(* Logix 5000 project; controller R1USB70001_CWRU_GRID_20120217 vendor 1 type 14 code 54 rev 19.11; software revision 19.01; part 2 of 3 *)
(* tags used below, declared in another part *)
   COM_TO_GRID_CLOSE_FAIL : BOOL;
   COM_TO_GRID_CLOSE_FAIL_THRESH : REAL;
   COM_TO_GRID_CLOSE_PROXY : BOOL;
   COM_TO_GRID_CLOSED : BOOL;
   COM_TO_GRID_COMMAND_CHANGED : BOOL;
   COM_TO_GRID_COMMAND_CHANGED_TIMER : TIMER;
   COM_TO_GRID_CURRENT : REAL;
   COM_TO_GRID_INT_REQ_CLOSE : BOOL;
   COM_TO_GRID_INT_REQ_CONNECT : BOOL;
   COM_TO_GRID_OPEN_FAIL : BOOL;
   COM_TO_GRID_OPEN_FAIL_THRESH : REAL;
   COM_TO_GRID_REQ_CLOSE : BOOL;
   COM_TO_GRID_REQ_CONNECT : BOOL;
   COM_TO_GRID_REQ_DISCONNECT : BOOL;
   COM_TO_GRID_REQ_OPEN : BOOL;
   COM_TO_SC_CLOSE_FAIL : BOOL;
   COM_TO_SC_CLOSE_FAIL_THRESH : REAL;
   COM_TO_SC_CLOSE_PROXY : BOOL;
   COM_TO_SC_CLOSED : BOOL;
   COM_TO_SC_COMMAND_CHANGED : BOOL;
   COM_TO_SC_COMMAND_CHANGED_TIMER : TIMER;
   COM_TO_SC_INT_REQ_CLOSE : BOOL;
   COM_TO_SC_INT_REQ_CONNECT : BOOL;
   COM_TO_SC_OPEN_FAIL : BOOL;
   COM_TO_SC_OPEN_FAIL_THRESH : REAL;
   COM_TO_SC_REQ_CLOSE : BOOL;
   COM_TO_SC_REQ_CONNECT : BOOL;
   COM_TO_SC_REQ_DISCONNECT : BOOL;
   COM_TO_SC_REQ_OPEN : BOOL;
   COM_TO_SF_CLOSE_FAIL : BOOL;
   COM_TO_SF_CLOSE_FAIL_THRESH : REAL;
   COM_TO_SF_CLOSE_PROXY : BOOL;
   COM_TO_SF_CLOSED : BOOL;
   COM_TO_SF_COMMAND_CHANGED : BOOL;
   COM_TO_SF_COMMAND_CHANGED_TIMER : TIMER;
   COM_TO_SF_INT_REQ_CLOSE : BOOL;
   COM_TO_SF_INT_REQ_CONNECT : BOOL;
   COM_TO_SF_OPEN_FAIL : BOOL;
   COM_TO_SF_OPEN_FAIL_THRESH : REAL;
   COM_TO_SF_REQ_CLOSE : BOOL;
   COM_TO_SF_REQ_CONNECT : BOOL;
   COM_TO_SF_REQ_DISCONNECT : BOOL;
   COM_TO_SF_REQ_OPEN : BOOL;
   COM_TO_WF_CLOSE_FAIL : BOOL;
   COM_TO_WF_CLOSE_FAIL_THRESH : REAL;
   COM_TO_WF_CLOSE_PROXY : BOOL;
   COM_TO_WF_CLOSED : BOOL;
   COM_TO_WF_COMMAND_CHANGED : BOOL;
   COM_TO_WF_COMMAND_CHANGED_TIMER : TIMER;
   COM_TO_WF_INT_REQ_CLOSE : BOOL;
   COM_TO_WF_INT_REQ_CONNECT : BOOL;
   COM_TO_WF_OPEN_FAIL : BOOL;
   COM_TO_WF_OPEN_FAIL_THRESH : REAL;
   COM_TO_WF_REQ_CLOSE : BOOL;
   COM_TO_WF_REQ_CONNECT : BOOL;
   COM_TO_WF_REQ_DISCONNECT : BOOL;
   COM_TO_WF_REQ_OPEN : BOOL;
   COM_TO_WT_CLOSE_FAIL : BOOL;
   COM_TO_WT_CLOSE_FAIL_THRESH : REAL;
   COM_TO_WT_CLOSE_PROXY : BOOL;
   COM_TO_WT_CLOSED : BOOL;
   COM_TO_WT_COMMAND_CHANGED : BOOL;
   COM_TO_WT_COMMAND_CHANGED_TIMER : TIMER;
   COM_TO_WT_INT_REQ_CLOSE : BOOL;
   COM_TO_WT_INT_REQ_CONNECT : BOOL;
   COM_TO_WT_OPEN_FAIL : BOOL;
   COM_TO_WT_OPEN_FAIL_THRESH : REAL;
   COM_TO_WT_REQ_CLOSE : BOOL;
   COM_TO_WT_REQ_CONNECT : BOOL;
   COM_TO_WT_REQ_DISCONNECT : BOOL;
   COM_TO_WT_REQ_OPEN : BOOL;
   IND_TO_SC_CLOSE_FAIL : BOOL;
   IND_TO_SC_CLOSE_PROXY : BOOL;
   IND_TO_SC_CLOSED : BOOL;
   IND_TO_SC_COMMAND_CHANGED : BOOL;
   IND_TO_SC_COMMAND_CHANGED_TIMER : TIMER;
   IND_TO_SC_INT_REQ_CLOSE : BOOL;
   IND_TO_SC_INT_REQ_CONNECT : BOOL;
   IND_TO_SC_OPEN_FAIL : BOOL;
   IND_TO_SC_REQ_CLOSE : BOOL;
   IND_TO_SC_REQ_CONNECT : BOOL;
   IND_TO_SC_REQ_DISCONNECT : BOOL;
   IND_TO_SC_REQ_OPEN : BOOL;
   IND_TO_SF_CLOSE_FAIL : BOOL;
   IND_TO_SF_CLOSE_FAIL_THRESH : REAL;
   IND_TO_SF_CLOSE_PROXY : BOOL;
   IND_TO_SF_CLOSED : BOOL;
   IND_TO_SF_COMMAND_CHANGED : BOOL;
   IND_TO_SF_COMMAND_CHANGED_TIMER : TIMER;
   IND_TO_SF_INT_REQ_CLOSE : BOOL;
   IND_TO_SF_INT_REQ_CONNECT : BOOL;
   IND_TO_SF_OPEN_FAIL : BOOL;
   IND_TO_SF_OPEN_FAIL_THRESH : REAL;
   IND_TO_SF_REQ_CLOSE : BOOL;
   IND_TO_SF_REQ_CONNECT : BOOL;
   IND_TO_SF_REQ_DISCONNECT : BOOL;
   IND_TO_SF_REQ_OPEN : BOOL;
   IND_TO_WT_CLOSE_FAIL : BOOL;
   IND_TO_WT_CLOSE_FAIL_THRESH : REAL;
   IND_TO_WT_CLOSED : BOOL;
   IND_TO_WT_COMMAND_CHANGED : BOOL;
   IND_TO_WT_COMMAND_CHANGED_TIMER : TIMER;
   IND_TO_WT_INT_REQ_CONNECT : BOOL;
   IND_TO_WT_OPEN_FAIL : BOOL;
   IND_TO_WT_OPEN_FAIL_THRESH : REAL;
   IND_TO_WT_REQ_CLOSE : BOOL;
   IND_TO_WT_REQ_CONNECT : BOOL;
   IND_TO_WT_REQ_OPEN : BOOL;
   SC_TO_COM_CURRENT : REAL;
   SC_TO_GRID_CLOSE_FAIL : BOOL;
   SC_TO_GRID_CLOSE_FAIL_THRESH : REAL;
   SC_TO_GRID_CLOSE_PROXY : BOOL;
   SC_TO_GRID_CLOSED : BOOL;
   SC_TO_GRID_COMMAND_CHANGED : BOOL;
   SC_TO_GRID_COMMAND_CHANGED_TIMER : TIMER;
   SC_TO_GRID_CURRENT : REAL;
   SC_TO_GRID_INT_REQ_CLOSE : BOOL;
   SC_TO_GRID_INT_REQ_CONNECT : BOOL;
   SC_TO_GRID_OPEN_FAIL : BOOL;
   SC_TO_GRID_OPEN_FAIL_THRESH : REAL;
   SC_TO_GRID_REQ_CLOSE : BOOL;
   SC_TO_GRID_REQ_CONNECT : BOOL;
   SC_TO_GRID_REQ_DISCONNECT : BOOL;
   SC_TO_GRID_REQ_OPEN : BOOL;
   SC_TO_IND_CLOSE_FAIL_THRESH : REAL;
   SC_TO_IND_CURRENT : REAL;
   SC_TO_IND_OPEN_FAIL_THRESH : REAL;
   SF_TO_COM_CURRENT : REAL;
   SF_TO_GRID_CLOSE_FAIL : BOOL;
   SF_TO_GRID_CLOSE_FAIL_THRESH : REAL;
   SF_TO_GRID_CLOSE_PROXY : BOOL;
   SF_TO_GRID_CLOSED : BOOL;
   SF_TO_GRID_COMMAND_CHANGED : BOOL;
   SF_TO_GRID_COMMAND_CHANGED_TIMER : TIMER;
   SF_TO_GRID_CURRENT : REAL;
   SF_TO_GRID_INT_REQ_CLOSE : BOOL;
   SF_TO_GRID_INT_REQ_CONNECT : BOOL;
   SF_TO_GRID_OPEN_FAIL : BOOL;
   SF_TO_GRID_OPEN_FAIL_THRESH : REAL;
   SF_TO_GRID_REQ_CLOSE : BOOL;
   SF_TO_GRID_REQ_CONNECT : BOOL;
   SF_TO_GRID_REQ_DISCONNECT : BOOL;
   SF_TO_GRID_REQ_OPEN : BOOL;
   SF_TO_IND_CURRENT : REAL;
   WF_TO_COM_CURRENT : REAL;
   WF_TO_GRID_CLOSE_FAIL : BOOL;
   WF_TO_GRID_CLOSE_FAIL_THRESH : REAL;
   WF_TO_GRID_CLOSE_PROXY : BOOL;
   WF_TO_GRID_CLOSED : BOOL;
   WF_TO_GRID_COMMAND_CHANGED : BOOL;
   WF_TO_GRID_COMMAND_CHANGED_TIMER : TIMER;
   WF_TO_GRID_CURRENT : REAL;
   WF_TO_GRID_INT_REQ_CLOSE : BOOL;
   WF_TO_GRID_INT_REQ_CONNECT : BOOL;
   WF_TO_GRID_OPEN_FAIL : BOOL;
   WF_TO_GRID_OPEN_FAIL_THRESH : REAL;
   WF_TO_GRID_REQ_CLOSE : BOOL;
   WF_TO_GRID_REQ_CONNECT : BOOL;
   WF_TO_GRID_REQ_DISCONNECT : BOOL;
   WF_TO_GRID_REQ_OPEN : BOOL;
   WT_TO_COM_CURRENT : REAL;
   WT_TO_GRID_CLOSE_FAIL : BOOL;
   WT_TO_GRID_CLOSE_FAIL_THRESH : REAL;
   WT_TO_GRID_CLOSE_PROXY : BOOL;
   WT_TO_GRID_CLOSED : BOOL;
   WT_TO_GRID_COMMAND_CHANGED : BOOL;
   WT_TO_GRID_COMMAND_CHANGED_TIMER : TIMER;
   WT_TO_GRID_CURRENT : REAL;
   WT_TO_GRID_INT_REQ_CLOSE : BOOL;
   WT_TO_GRID_INT_REQ_CONNECT : BOOL;
   WT_TO_GRID_OPEN_FAIL : BOOL;
   WT_TO_GRID_OPEN_FAIL_THRESH : REAL;
   WT_TO_GRID_REQ_CLOSE : BOOL;
   WT_TO_GRID_REQ_CONNECT : BOOL;
   WT_TO_GRID_REQ_DISCONNECT : BOOL;
   WT_TO_GRID_REQ_OPEN : BOOL;
   WT_TO_IND_CURRENT : REAL;
   CL_GP_GD_CS : ALIAS FOR ACNR_GP_SC_N2:15:O.1;
   CL_GP_SC_CS : ALIAS FOR ACNR_GP_SC_N2:15:O.5;
   CL_GP_SF_CS : ALIAS FOR ACNR_GP_SC_N2:15:O.4;
   CL_GP_WF_CS : ALIAS FOR ACNR_GP_SC_N2:15:O.2;
   CL_GP_WT_CS : ALIAS FOR ACNR_GP_SC_N2:15:O.3;
   IL_GP_SC_CS : ALIAS FOR ACNR_GP_SC_N2:16:O.2;
   IL_GP_SF_CS : ALIAS FOR ACNR_GP_SC_N2:16:O.1;
   SC_GP_GD_CS : ALIAS FOR ACNR_GP_SC_N2:14:O.2;
   SF_GP_GD_CS : ALIAS FOR ACNR_GP_SC_N2:14:O.0;
   WF_GP_GD_CS : ALIAS FOR ACNR_GP_SC_N2:13:O.3;
   WT_GP_GD_CS : ALIAS FOR ACNR_GP_SC_N2:13:O.5;
(* MainProgram, continued *)

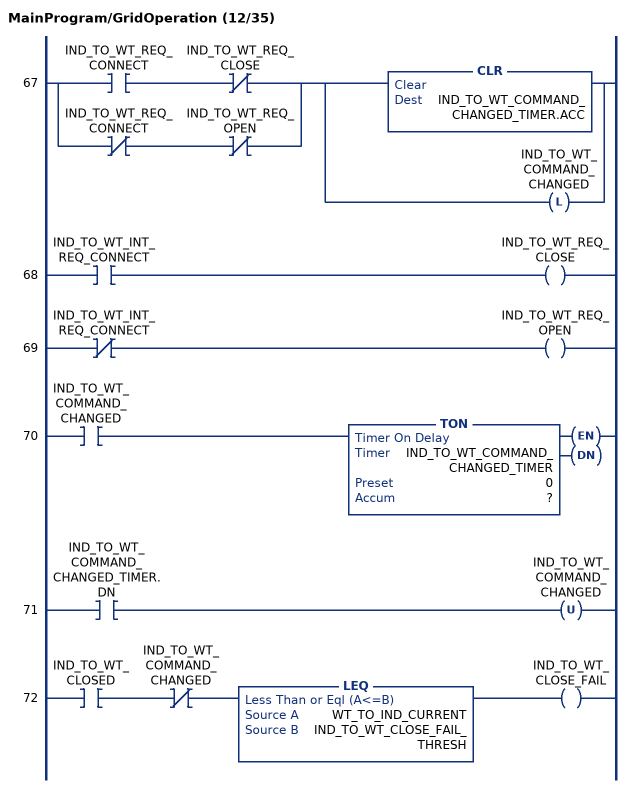
   [picture p24: MainProgram/GridOperation rungs 67-72]
   67: [XIC(IND_TO_WT_REQ_CONNECT) XIO(IND_TO_WT_REQ_CLOSE) ,XIO(IND_TO_WT_REQ_CONNECT) XIO(IND_TO_WT_REQ_OPEN) ][CLR(IND_TO_WT_COMMAND_CHANGED_TIMER.ACC) ,OTL(IND_TO_WT_COMMAND_CHANGED) ];
   68: XIC(IND_TO_WT_INT_REQ_CONNECT)OTE(IND_TO_WT_REQ_CLOSE);
   69: XIO(IND_TO_WT_INT_REQ_CONNECT)OTE(IND_TO_WT_REQ_OPEN);
   70: XIC(IND_TO_WT_COMMAND_CHANGED)TON(IND_TO_WT_COMMAND_CHANGED_TIMER,?,?);
   71: XIC(IND_TO_WT_COMMAND_CHANGED_TIMER.DN)OTU(IND_TO_WT_COMMAND_CHANGED);
   72: XIC(IND_TO_WT_CLOSED)XIO(IND_TO_WT_COMMAND_CHANGED)LEQ(WT_TO_IND_CURRENT,IND_TO_WT_CLOSE_FAIL_THRESH)OTE(IND_TO_WT_CLOSE_FAIL);
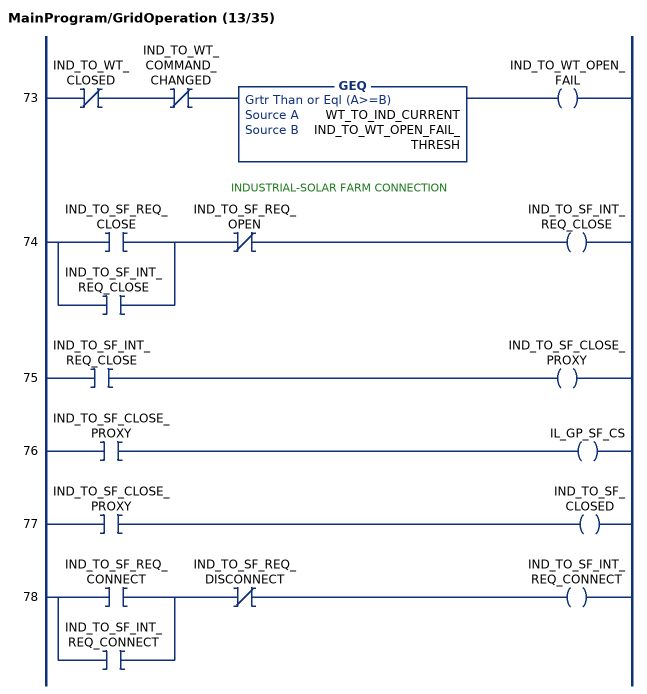
   73: XIO(IND_TO_WT_CLOSED)XIO(IND_TO_WT_COMMAND_CHANGED)GEQ(WT_TO_IND_CURRENT,IND_TO_WT_OPEN_FAIL_THRESH)OTE(IND_TO_WT_OPEN_FAIL);
   // INDUSTRIAL-SOLAR FARM CONNECTION
   74: [XIC(IND_TO_SF_REQ_CLOSE) ,XIC(IND_TO_SF_INT_REQ_CLOSE) ]XIO(IND_TO_SF_REQ_OPEN)OTE(IND_TO_SF_INT_REQ_CLOSE);
   75: XIC(IND_TO_SF_INT_REQ_CLOSE)OTE(IND_TO_SF_CLOSE_PROXY);
   76: XIC(IND_TO_SF_CLOSE_PROXY)OTE(IL_GP_SF_CS);
   77: XIC(IND_TO_SF_CLOSE_PROXY)OTE(IND_TO_SF_CLOSED);
   78: [XIC(IND_TO_SF_REQ_CONNECT) ,XIC(IND_TO_SF_INT_REQ_CONNECT) ]XIO(IND_TO_SF_REQ_DISCONNECT)OTE(IND_TO_SF_INT_REQ_CONNECT);
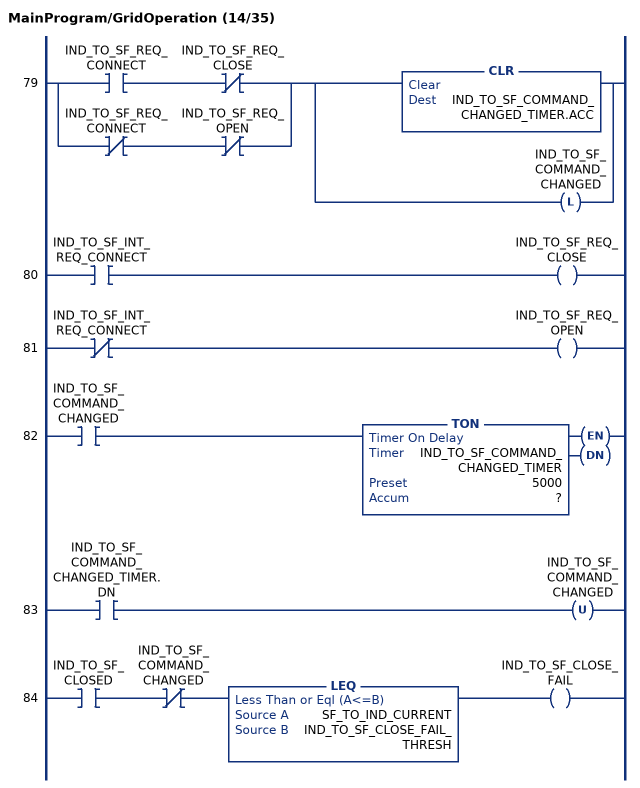
   79: [XIC(IND_TO_SF_REQ_CONNECT) XIO(IND_TO_SF_REQ_CLOSE) ,XIO(IND_TO_SF_REQ_CONNECT) XIO(IND_TO_SF_REQ_OPEN) ][CLR(IND_TO_SF_COMMAND_CHANGED_TIMER.ACC) ,OTL(IND_TO_SF_COMMAND_CHANGED) ];
   80: XIC(IND_TO_SF_INT_REQ_CONNECT)OTE(IND_TO_SF_REQ_CLOSE);
   81: XIO(IND_TO_SF_INT_REQ_CONNECT)OTE(IND_TO_SF_REQ_OPEN);
   82: XIC(IND_TO_SF_COMMAND_CHANGED)TON(IND_TO_SF_COMMAND_CHANGED_TIMER,?,?);
   83: XIC(IND_TO_SF_COMMAND_CHANGED_TIMER.DN)OTU(IND_TO_SF_COMMAND_CHANGED);
   84: XIC(IND_TO_SF_CLOSED)XIO(IND_TO_SF_COMMAND_CHANGED)LEQ(SF_TO_IND_CURRENT,IND_TO_SF_CLOSE_FAIL_THRESH)OTE(IND_TO_SF_CLOSE_FAIL);
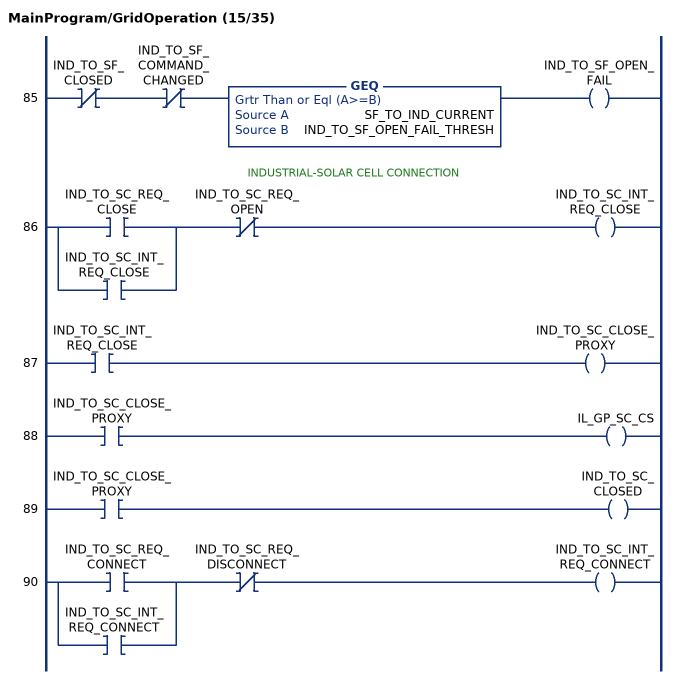
   85: XIO(IND_TO_SF_CLOSED)XIO(IND_TO_SF_COMMAND_CHANGED)GEQ(SF_TO_IND_CURRENT,IND_TO_SF_OPEN_FAIL_THRESH)OTE(IND_TO_SF_OPEN_FAIL);
   // INDUSTRIAL-SOLAR CELL CONNECTION
   86: [XIC(IND_TO_SC_REQ_CLOSE) ,XIC(IND_TO_SC_INT_REQ_CLOSE) ]XIO(IND_TO_SC_REQ_OPEN)OTE(IND_TO_SC_INT_REQ_CLOSE);
   87: XIC(IND_TO_SC_INT_REQ_CLOSE)OTE(IND_TO_SC_CLOSE_PROXY);
   88: XIC(IND_TO_SC_CLOSE_PROXY)OTE(IL_GP_SC_CS);
   89: XIC(IND_TO_SC_CLOSE_PROXY)OTE(IND_TO_SC_CLOSED);
   90: [XIC(IND_TO_SC_REQ_CONNECT) ,XIC(IND_TO_SC_INT_REQ_CONNECT) ]XIO(IND_TO_SC_REQ_DISCONNECT)OTE(IND_TO_SC_INT_REQ_CONNECT);
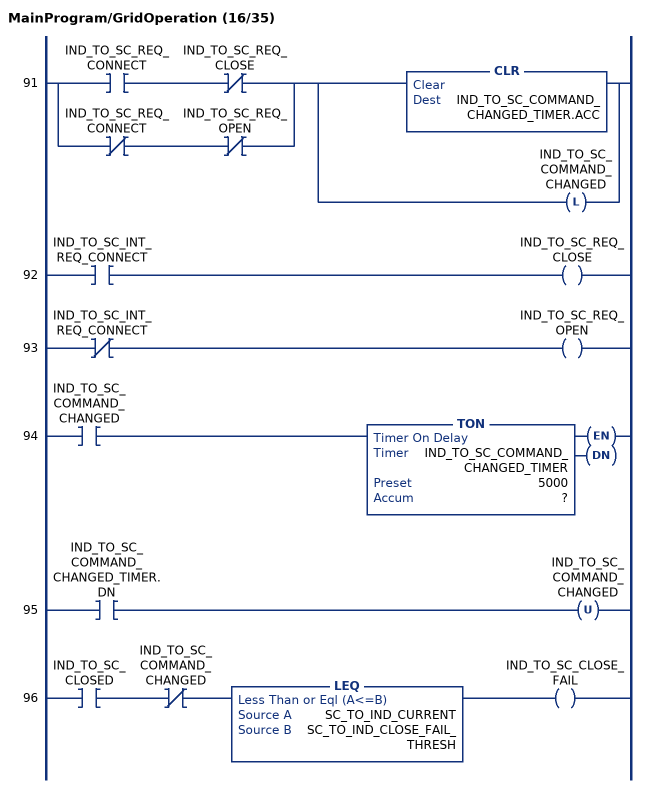
   91: [XIC(IND_TO_SC_REQ_CONNECT) XIO(IND_TO_SC_REQ_CLOSE) ,XIO(IND_TO_SC_REQ_CONNECT) XIO(IND_TO_SC_REQ_OPEN) ][CLR(IND_TO_SC_COMMAND_CHANGED_TIMER.ACC) ,OTL(IND_TO_SC_COMMAND_CHANGED) ];
   92: XIC(IND_TO_SC_INT_REQ_CONNECT)OTE(IND_TO_SC_REQ_CLOSE);
   93: XIO(IND_TO_SC_INT_REQ_CONNECT)OTE(IND_TO_SC_REQ_OPEN);
   94: XIC(IND_TO_SC_COMMAND_CHANGED)TON(IND_TO_SC_COMMAND_CHANGED_TIMER,?,?);
   95: XIC(IND_TO_SC_COMMAND_CHANGED_TIMER.DN)OTU(IND_TO_SC_COMMAND_CHANGED);
   96: XIC(IND_TO_SC_CLOSED)XIO(IND_TO_SC_COMMAND_CHANGED)LEQ(SC_TO_IND_CURRENT,SC_TO_IND_CLOSE_FAIL_THRESH)OTE(IND_TO_SC_CLOSE_FAIL);
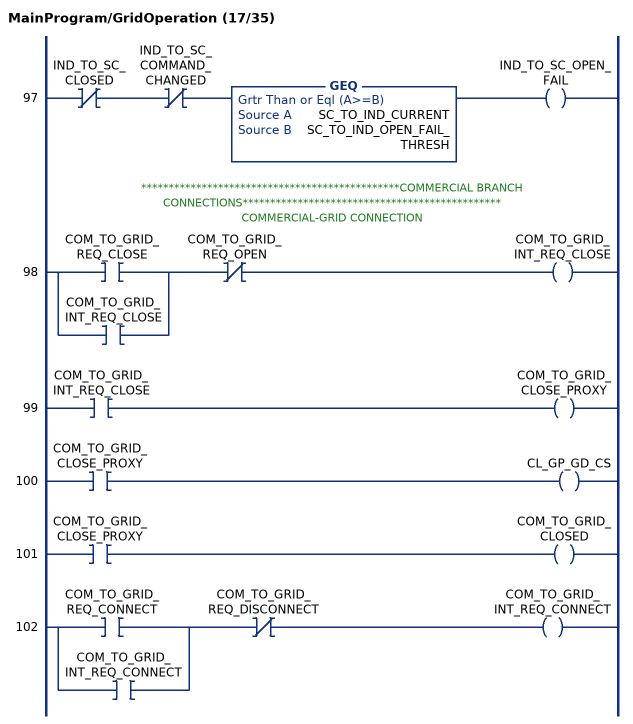
   97: XIO(IND_TO_SC_CLOSED)XIO(IND_TO_SC_COMMAND_CHANGED)GEQ(SC_TO_IND_CURRENT,SC_TO_IND_OPEN_FAIL_THRESH)OTE(IND_TO_SC_OPEN_FAIL);
   // ***********************************************COMMERCIAL BRANCH CONNECTIONS***********************************************
   // COMMERCIAL-GRID CONNECTION
   98: [XIC(COM_TO_GRID_REQ_CLOSE) ,XIC(COM_TO_GRID_INT_REQ_CLOSE) ]XIO(COM_TO_GRID_REQ_OPEN)OTE(COM_TO_GRID_INT_REQ_CLOSE);
   99: XIC(COM_TO_GRID_INT_REQ_CLOSE)OTE(COM_TO_GRID_CLOSE_PROXY);
   100: XIC(COM_TO_GRID_CLOSE_PROXY)OTE(CL_GP_GD_CS);
   101: XIC(COM_TO_GRID_CLOSE_PROXY)OTE(COM_TO_GRID_CLOSED);
   102: [XIC(COM_TO_GRID_REQ_CONNECT) ,XIC(COM_TO_GRID_INT_REQ_CONNECT) ]XIO(COM_TO_GRID_REQ_DISCONNECT)OTE(COM_TO_GRID_INT_REQ_CONNECT);
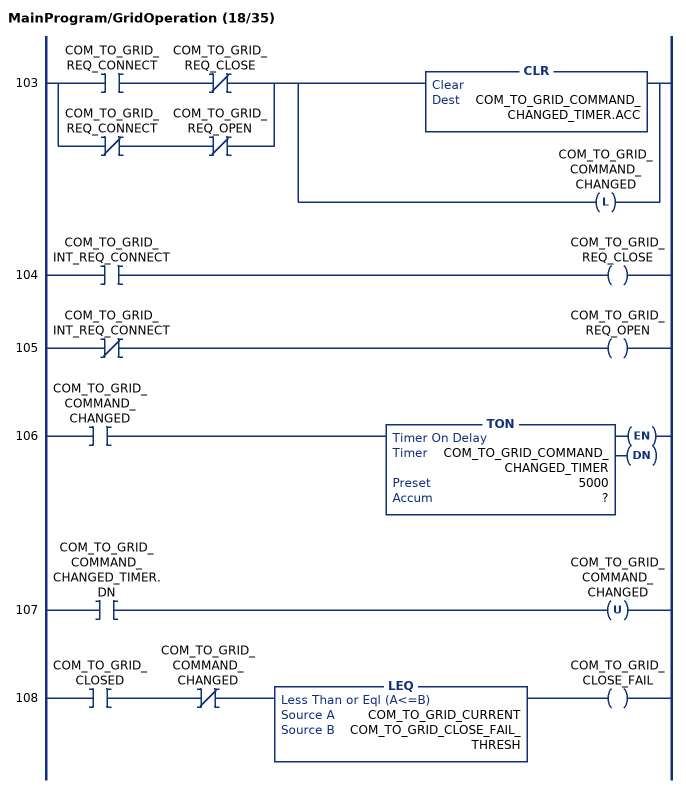
   103: [XIC(COM_TO_GRID_REQ_CONNECT) XIO(COM_TO_GRID_REQ_CLOSE) ,XIO(COM_TO_GRID_REQ_CONNECT) XIO(COM_TO_GRID_REQ_OPEN) ][CLR(COM_TO_GRID_COMMAND_CHANGED_TIMER.ACC) ,OTL(COM_TO_GRID_COMMAND_CHANGED) ];
   104: XIC(COM_TO_GRID_INT_REQ_CONNECT)OTE(COM_TO_GRID_REQ_CLOSE);
   105: XIO(COM_TO_GRID_INT_REQ_CONNECT)OTE(COM_TO_GRID_REQ_OPEN);
   106: XIC(COM_TO_GRID_COMMAND_CHANGED)TON(COM_TO_GRID_COMMAND_CHANGED_TIMER,?,?);
   107: XIC(COM_TO_GRID_COMMAND_CHANGED_TIMER.DN)OTU(COM_TO_GRID_COMMAND_CHANGED);
   108: XIC(COM_TO_GRID_CLOSED)XIO(COM_TO_GRID_COMMAND_CHANGED)LEQ(COM_TO_GRID_CURRENT,COM_TO_GRID_CLOSE_FAIL_THRESH)OTE(COM_TO_GRID_CLOSE_FAIL);
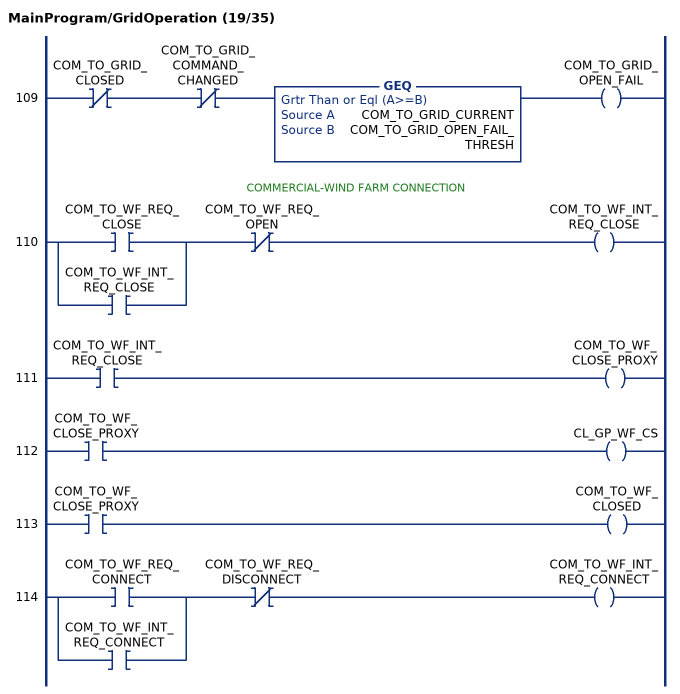
   109: XIO(COM_TO_GRID_CLOSED)XIO(COM_TO_GRID_COMMAND_CHANGED)GEQ(COM_TO_GRID_CURRENT,COM_TO_GRID_OPEN_FAIL_THRESH)OTE(COM_TO_GRID_OPEN_FAIL);
   // COMMERCIAL-WIND FARM CONNECTION
   110: [XIC(COM_TO_WF_REQ_CLOSE) ,XIC(COM_TO_WF_INT_REQ_CLOSE) ]XIO(COM_TO_WF_REQ_OPEN)OTE(COM_TO_WF_INT_REQ_CLOSE);
   111: XIC(COM_TO_WF_INT_REQ_CLOSE)OTE(COM_TO_WF_CLOSE_PROXY);
   112: XIC(COM_TO_WF_CLOSE_PROXY)OTE(CL_GP_WF_CS);
   113: XIC(COM_TO_WF_CLOSE_PROXY)OTE(COM_TO_WF_CLOSED);
   114: [XIC(COM_TO_WF_REQ_CONNECT) ,XIC(COM_TO_WF_INT_REQ_CONNECT) ]XIO(COM_TO_WF_REQ_DISCONNECT)OTE(COM_TO_WF_INT_REQ_CONNECT);
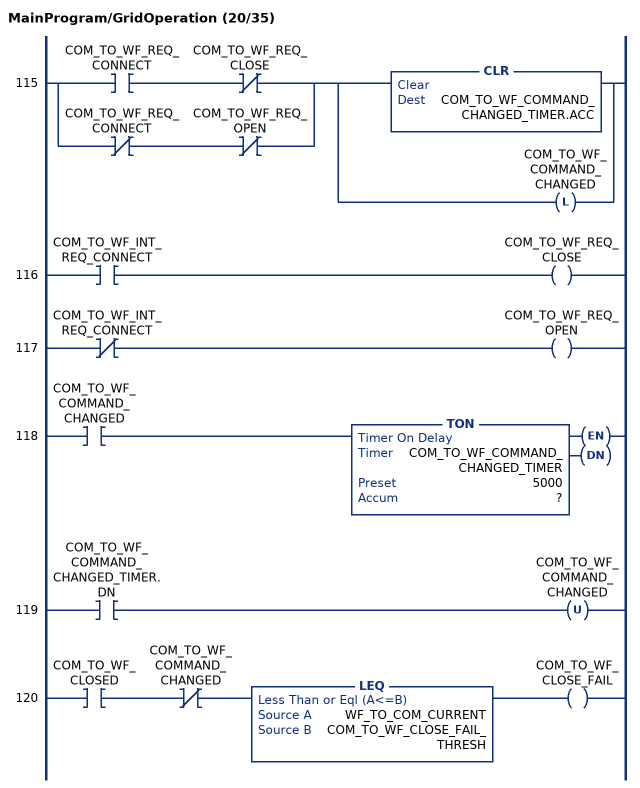
   115: [XIC(COM_TO_WF_REQ_CONNECT) XIO(COM_TO_WF_REQ_CLOSE) ,XIO(COM_TO_WF_REQ_CONNECT) XIO(COM_TO_WF_REQ_OPEN) ][CLR(COM_TO_WF_COMMAND_CHANGED_TIMER.ACC) ,OTL(COM_TO_WF_COMMAND_CHANGED) ];
   116: XIC(COM_TO_WF_INT_REQ_CONNECT)OTE(COM_TO_WF_REQ_CLOSE);
   117: XIO(COM_TO_WF_INT_REQ_CONNECT)OTE(COM_TO_WF_REQ_OPEN);
   118: XIC(COM_TO_WF_COMMAND_CHANGED)TON(COM_TO_WF_COMMAND_CHANGED_TIMER,?,?);
   119: XIC(COM_TO_WF_COMMAND_CHANGED_TIMER.DN)OTU(COM_TO_WF_COMMAND_CHANGED);
   120: XIC(COM_TO_WF_CLOSED)XIO(COM_TO_WF_COMMAND_CHANGED)LEQ(WF_TO_COM_CURRENT,COM_TO_WF_CLOSE_FAIL_THRESH)OTE(COM_TO_WF_CLOSE_FAIL);
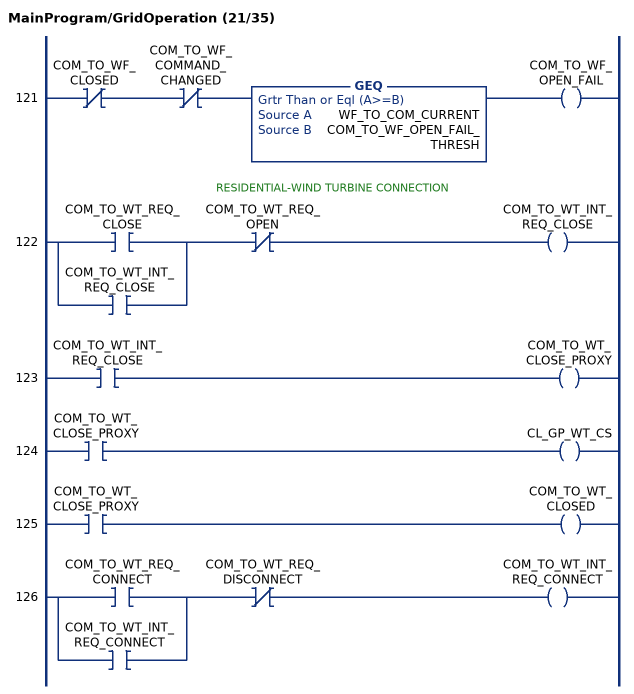
   121: XIO(COM_TO_WF_CLOSED)XIO(COM_TO_WF_COMMAND_CHANGED)GEQ(WF_TO_COM_CURRENT,COM_TO_WF_OPEN_FAIL_THRESH)OTE(COM_TO_WF_OPEN_FAIL);
   // RESIDENTIAL-WIND TURBINE CONNECTION
   122: [XIC(COM_TO_WT_REQ_CLOSE) ,XIC(COM_TO_WT_INT_REQ_CLOSE) ]XIO(COM_TO_WT_REQ_OPEN)OTE(COM_TO_WT_INT_REQ_CLOSE);
   123: XIC(COM_TO_WT_INT_REQ_CLOSE)OTE(COM_TO_WT_CLOSE_PROXY);
   124: XIC(COM_TO_WT_CLOSE_PROXY)OTE(CL_GP_WT_CS);
   125: XIC(COM_TO_WT_CLOSE_PROXY)OTE(COM_TO_WT_CLOSED);
   126: [XIC(COM_TO_WT_REQ_CONNECT) ,XIC(COM_TO_WT_INT_REQ_CONNECT) ]XIO(COM_TO_WT_REQ_DISCONNECT)OTE(COM_TO_WT_INT_REQ_CONNECT);
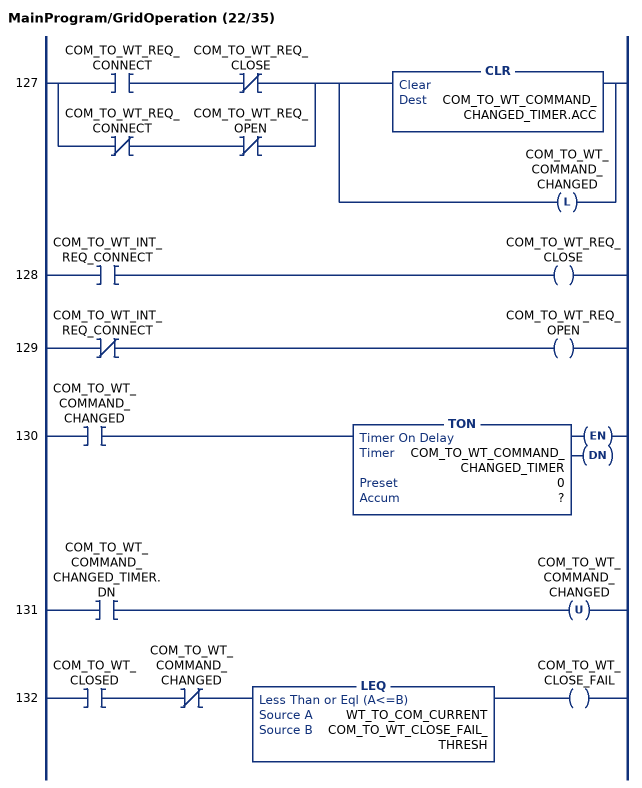
   127: [XIC(COM_TO_WT_REQ_CONNECT) XIO(COM_TO_WT_REQ_CLOSE) ,XIO(COM_TO_WT_REQ_CONNECT) XIO(COM_TO_WT_REQ_OPEN) ][CLR(COM_TO_WT_COMMAND_CHANGED_TIMER.ACC) ,OTL(COM_TO_WT_COMMAND_CHANGED) ];
   128: XIC(COM_TO_WT_INT_REQ_CONNECT)OTE(COM_TO_WT_REQ_CLOSE);
   129: XIO(COM_TO_WT_INT_REQ_CONNECT)OTE(COM_TO_WT_REQ_OPEN);
   130: XIC(COM_TO_WT_COMMAND_CHANGED)TON(COM_TO_WT_COMMAND_CHANGED_TIMER,?,?);
   131: XIC(COM_TO_WT_COMMAND_CHANGED_TIMER.DN)OTU(COM_TO_WT_COMMAND_CHANGED);
   132: XIC(COM_TO_WT_CLOSED)XIO(COM_TO_WT_COMMAND_CHANGED)LEQ(WT_TO_COM_CURRENT,COM_TO_WT_CLOSE_FAIL_THRESH)OTE(COM_TO_WT_CLOSE_FAIL);
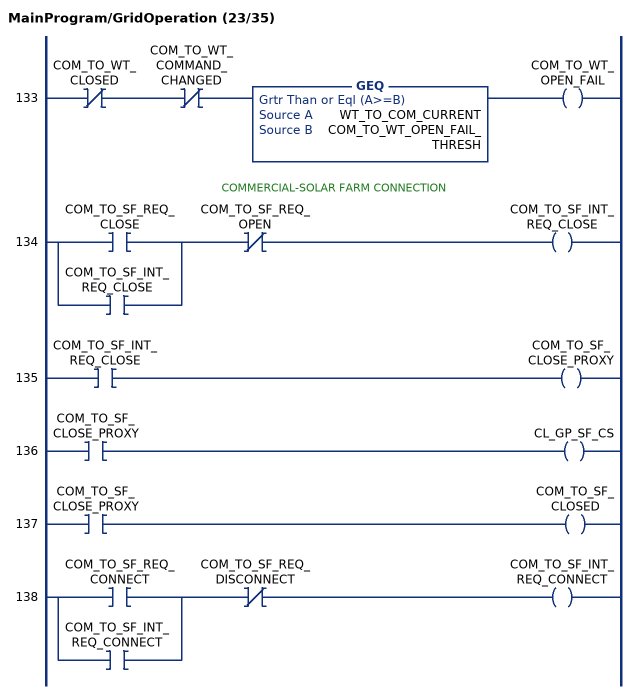
   133: XIO(COM_TO_WT_CLOSED)XIO(COM_TO_WT_COMMAND_CHANGED)GEQ(WT_TO_COM_CURRENT,COM_TO_WT_OPEN_FAIL_THRESH)OTE(COM_TO_WT_OPEN_FAIL);
   // COMMERCIAL-SOLAR FARM CONNECTION
   134: [XIC(COM_TO_SF_REQ_CLOSE) ,XIC(COM_TO_SF_INT_REQ_CLOSE) ]XIO(COM_TO_SF_REQ_OPEN)OTE(COM_TO_SF_INT_REQ_CLOSE);
   135: XIC(COM_TO_SF_INT_REQ_CLOSE)OTE(COM_TO_SF_CLOSE_PROXY);
   136: XIC(COM_TO_SF_CLOSE_PROXY)OTE(CL_GP_SF_CS);
   137: XIC(COM_TO_SF_CLOSE_PROXY)OTE(COM_TO_SF_CLOSED);
   138: [XIC(COM_TO_SF_REQ_CONNECT) ,XIC(COM_TO_SF_INT_REQ_CONNECT) ]XIO(COM_TO_SF_REQ_DISCONNECT)OTE(COM_TO_SF_INT_REQ_CONNECT);
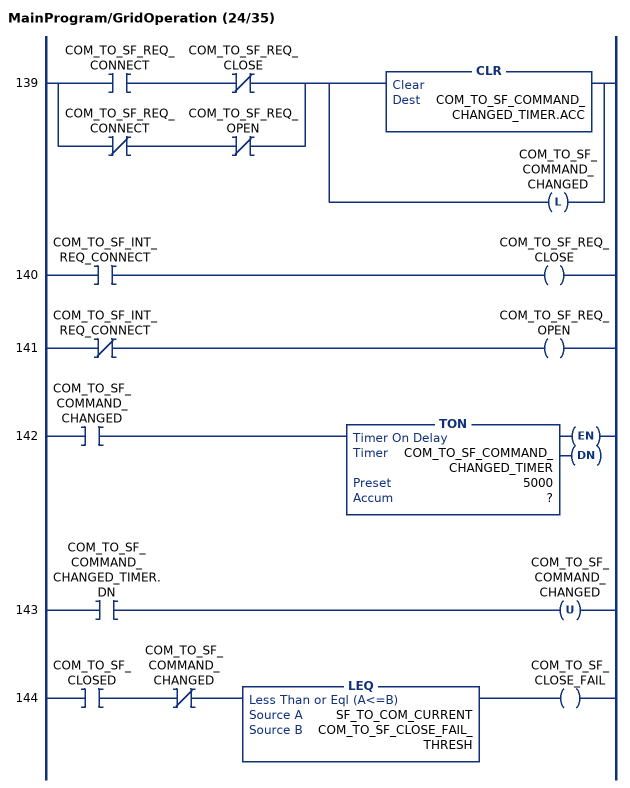
   139: [XIC(COM_TO_SF_REQ_CONNECT) XIO(COM_TO_SF_REQ_CLOSE) ,XIO(COM_TO_SF_REQ_CONNECT) XIO(COM_TO_SF_REQ_OPEN) ][CLR(COM_TO_SF_COMMAND_CHANGED_TIMER.ACC) ,OTL(COM_TO_SF_COMMAND_CHANGED) ];
   140: XIC(COM_TO_SF_INT_REQ_CONNECT)OTE(COM_TO_SF_REQ_CLOSE);
   141: XIO(COM_TO_SF_INT_REQ_CONNECT)OTE(COM_TO_SF_REQ_OPEN);
   142: XIC(COM_TO_SF_COMMAND_CHANGED)TON(COM_TO_SF_COMMAND_CHANGED_TIMER,?,?);
   143: XIC(COM_TO_SF_COMMAND_CHANGED_TIMER.DN)OTU(COM_TO_SF_COMMAND_CHANGED);
   144: XIC(COM_TO_SF_CLOSED)XIO(COM_TO_SF_COMMAND_CHANGED)LEQ(SF_TO_COM_CURRENT,COM_TO_SF_CLOSE_FAIL_THRESH)OTE(COM_TO_SF_CLOSE_FAIL);
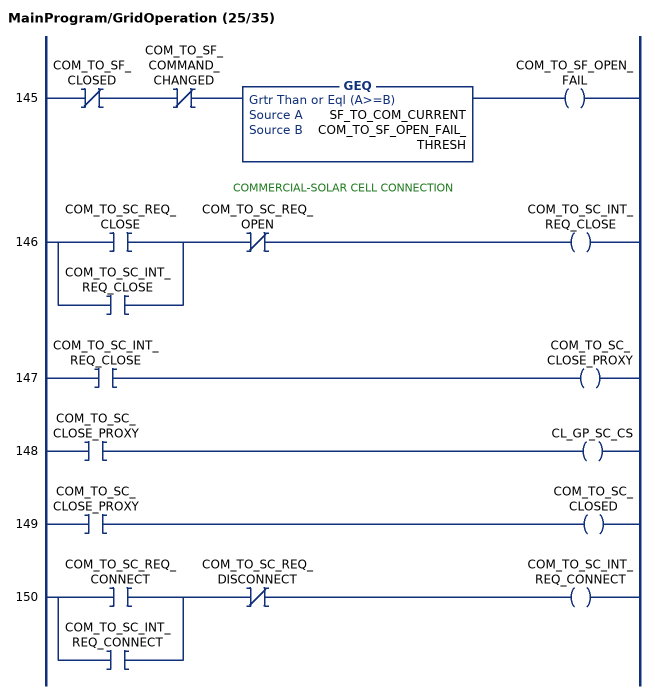
   145: XIO(COM_TO_SF_CLOSED)XIO(COM_TO_SF_COMMAND_CHANGED)GEQ(SF_TO_COM_CURRENT,COM_TO_SF_OPEN_FAIL_THRESH)OTE(COM_TO_SF_OPEN_FAIL);
   // COMMERCIAL-SOLAR CELL CONNECTION
   146: [XIC(COM_TO_SC_REQ_CLOSE) ,XIC(COM_TO_SC_INT_REQ_CLOSE) ]XIO(COM_TO_SC_REQ_OPEN)OTE(COM_TO_SC_INT_REQ_CLOSE);
   147: XIC(COM_TO_SC_INT_REQ_CLOSE)OTE(COM_TO_SC_CLOSE_PROXY);
   148: XIC(COM_TO_SC_CLOSE_PROXY)OTE(CL_GP_SC_CS);
   149: XIC(COM_TO_SC_CLOSE_PROXY)OTE(COM_TO_SC_CLOSED);
   150: [XIC(COM_TO_SC_REQ_CONNECT) ,XIC(COM_TO_SC_INT_REQ_CONNECT) ]XIO(COM_TO_SC_REQ_DISCONNECT)OTE(COM_TO_SC_INT_REQ_CONNECT);
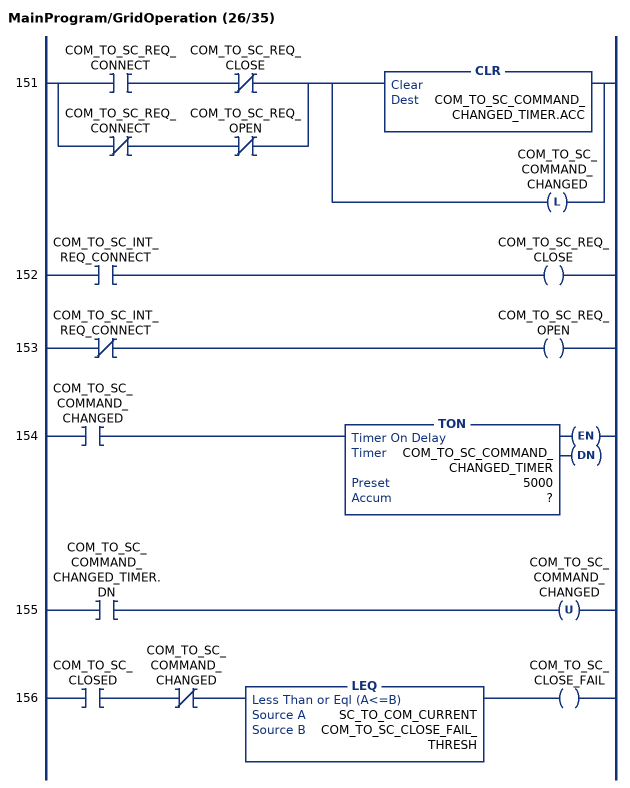
   151: [XIC(COM_TO_SC_REQ_CONNECT) XIO(COM_TO_SC_REQ_CLOSE) ,XIO(COM_TO_SC_REQ_CONNECT) XIO(COM_TO_SC_REQ_OPEN) ][CLR(COM_TO_SC_COMMAND_CHANGED_TIMER.ACC) ,OTL(COM_TO_SC_COMMAND_CHANGED) ];
   152: XIC(COM_TO_SC_INT_REQ_CONNECT)OTE(COM_TO_SC_REQ_CLOSE);
   153: XIO(COM_TO_SC_INT_REQ_CONNECT)OTE(COM_TO_SC_REQ_OPEN);
   154: XIC(COM_TO_SC_COMMAND_CHANGED)TON(COM_TO_SC_COMMAND_CHANGED_TIMER,?,?);
   155: XIC(COM_TO_SC_COMMAND_CHANGED_TIMER.DN)OTU(COM_TO_SC_COMMAND_CHANGED);
   156: XIC(COM_TO_SC_CLOSED)XIO(COM_TO_SC_COMMAND_CHANGED)LEQ(SC_TO_COM_CURRENT,COM_TO_SC_CLOSE_FAIL_THRESH)OTE(COM_TO_SC_CLOSE_FAIL);
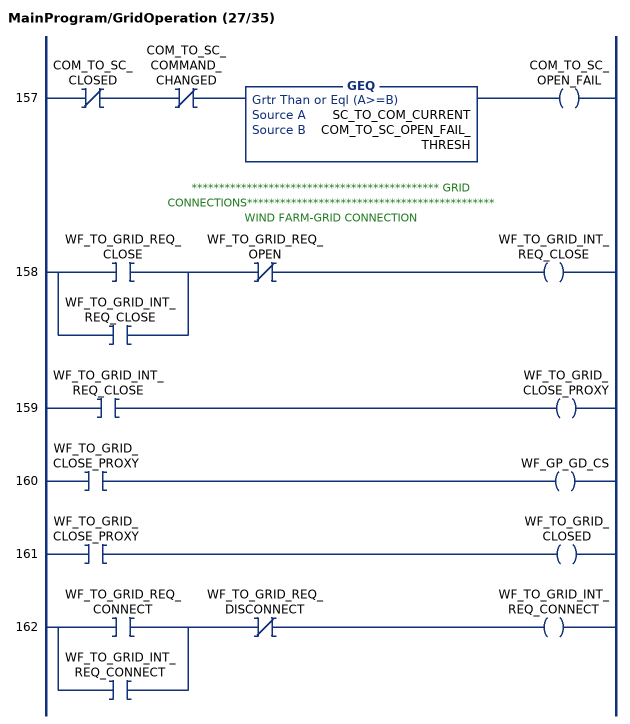
   157: XIO(COM_TO_SC_CLOSED)XIO(COM_TO_SC_COMMAND_CHANGED)GEQ(SC_TO_COM_CURRENT,COM_TO_SC_OPEN_FAIL_THRESH)OTE(COM_TO_SC_OPEN_FAIL);
   // ********************************************* GRID CONNECTIONS*********************************************
   // WIND FARM-GRID CONNECTION
   158: [XIC(WF_TO_GRID_REQ_CLOSE) ,XIC(WF_TO_GRID_INT_REQ_CLOSE) ]XIO(WF_TO_GRID_REQ_OPEN)OTE(WF_TO_GRID_INT_REQ_CLOSE);
   159: XIC(WF_TO_GRID_INT_REQ_CLOSE)OTE(WF_TO_GRID_CLOSE_PROXY);
   160: XIC(WF_TO_GRID_CLOSE_PROXY)OTE(WF_GP_GD_CS);
   161: XIC(WF_TO_GRID_CLOSE_PROXY)OTE(WF_TO_GRID_CLOSED);
   162: [XIC(WF_TO_GRID_REQ_CONNECT) ,XIC(WF_TO_GRID_INT_REQ_CONNECT) ]XIO(WF_TO_GRID_REQ_DISCONNECT)OTE(WF_TO_GRID_INT_REQ_CONNECT);
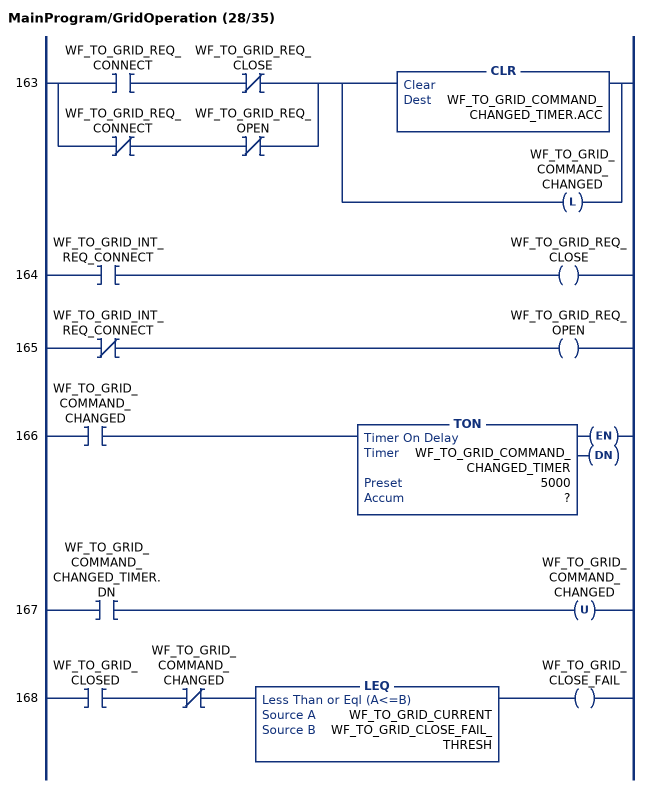
   163: [XIC(WF_TO_GRID_REQ_CONNECT) XIO(WF_TO_GRID_REQ_CLOSE) ,XIO(WF_TO_GRID_REQ_CONNECT) XIO(WF_TO_GRID_REQ_OPEN) ][CLR(WF_TO_GRID_COMMAND_CHANGED_TIMER.ACC) ,OTL(WF_TO_GRID_COMMAND_CHANGED) ];
   164: XIC(WF_TO_GRID_INT_REQ_CONNECT)OTE(WF_TO_GRID_REQ_CLOSE);
   165: XIO(WF_TO_GRID_INT_REQ_CONNECT)OTE(WF_TO_GRID_REQ_OPEN);
   166: XIC(WF_TO_GRID_COMMAND_CHANGED)TON(WF_TO_GRID_COMMAND_CHANGED_TIMER,?,?);
   167: XIC(WF_TO_GRID_COMMAND_CHANGED_TIMER.DN)OTU(WF_TO_GRID_COMMAND_CHANGED);
   168: XIC(WF_TO_GRID_CLOSED)XIO(WF_TO_GRID_COMMAND_CHANGED)LEQ(WF_TO_GRID_CURRENT,WF_TO_GRID_CLOSE_FAIL_THRESH)OTE(WF_TO_GRID_CLOSE_FAIL);
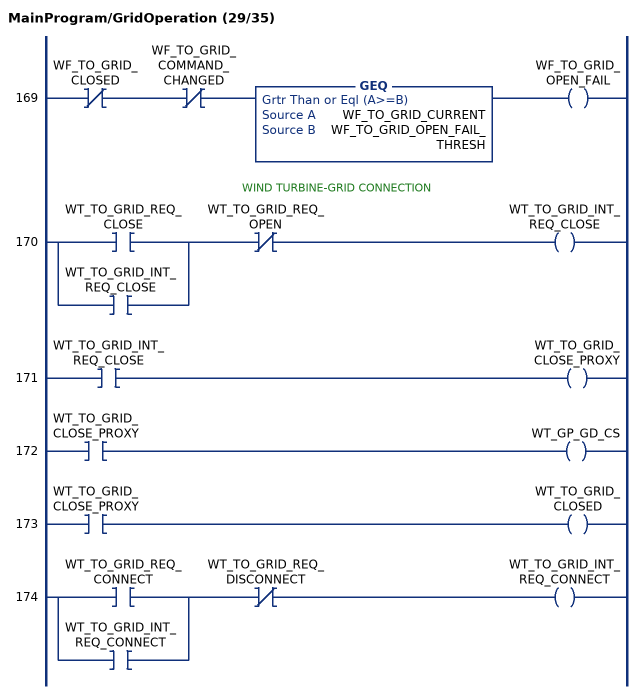
   169: XIO(WF_TO_GRID_CLOSED)XIO(WF_TO_GRID_COMMAND_CHANGED)GEQ(WF_TO_GRID_CURRENT,WF_TO_GRID_OPEN_FAIL_THRESH)OTE(WF_TO_GRID_OPEN_FAIL);
   // WIND TURBINE-GRID CONNECTION
   170: [XIC(WT_TO_GRID_REQ_CLOSE) ,XIC(WT_TO_GRID_INT_REQ_CLOSE) ]XIO(WT_TO_GRID_REQ_OPEN)OTE(WT_TO_GRID_INT_REQ_CLOSE);
   171: XIC(WT_TO_GRID_INT_REQ_CLOSE)OTE(WT_TO_GRID_CLOSE_PROXY);
   172: XIC(WT_TO_GRID_CLOSE_PROXY)OTE(WT_GP_GD_CS);
   173: XIC(WT_TO_GRID_CLOSE_PROXY)OTE(WT_TO_GRID_CLOSED);
   174: [XIC(WT_TO_GRID_REQ_CONNECT) ,XIC(WT_TO_GRID_INT_REQ_CONNECT) ]XIO(WT_TO_GRID_REQ_DISCONNECT)OTE(WT_TO_GRID_INT_REQ_CONNECT);
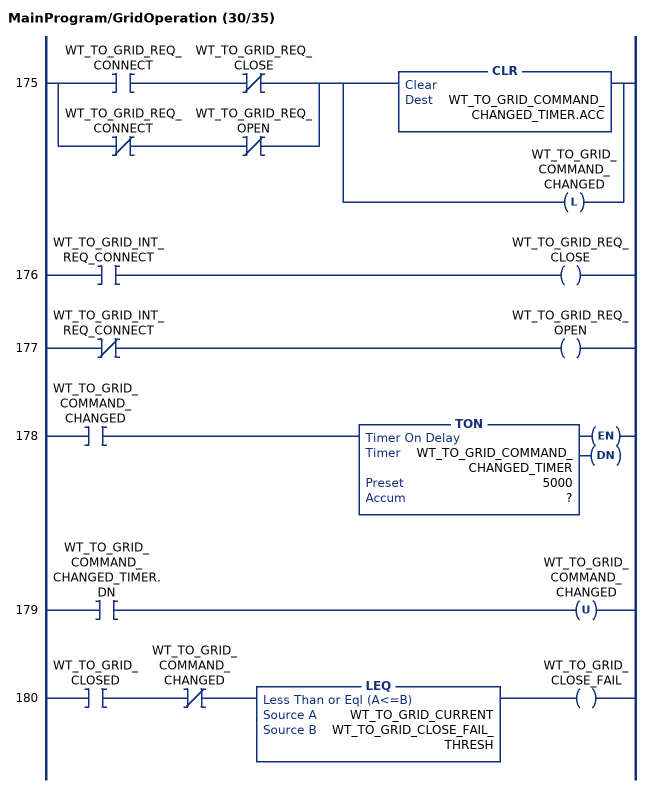
   175: [XIC(WT_TO_GRID_REQ_CONNECT) XIO(WT_TO_GRID_REQ_CLOSE) ,XIO(WT_TO_GRID_REQ_CONNECT) XIO(WT_TO_GRID_REQ_OPEN) ][CLR(WT_TO_GRID_COMMAND_CHANGED_TIMER.ACC) ,OTL(WT_TO_GRID_COMMAND_CHANGED) ];
   176: XIC(WT_TO_GRID_INT_REQ_CONNECT)OTE(WT_TO_GRID_REQ_CLOSE);
   177: XIO(WT_TO_GRID_INT_REQ_CONNECT)OTE(WT_TO_GRID_REQ_OPEN);
   178: XIC(WT_TO_GRID_COMMAND_CHANGED)TON(WT_TO_GRID_COMMAND_CHANGED_TIMER,?,?);
   179: XIC(WT_TO_GRID_COMMAND_CHANGED_TIMER.DN)OTU(WT_TO_GRID_COMMAND_CHANGED);
   180: XIC(WT_TO_GRID_CLOSED)XIO(WT_TO_GRID_COMMAND_CHANGED)LEQ(WT_TO_GRID_CURRENT,WT_TO_GRID_CLOSE_FAIL_THRESH)OTE(WT_TO_GRID_CLOSE_FAIL);
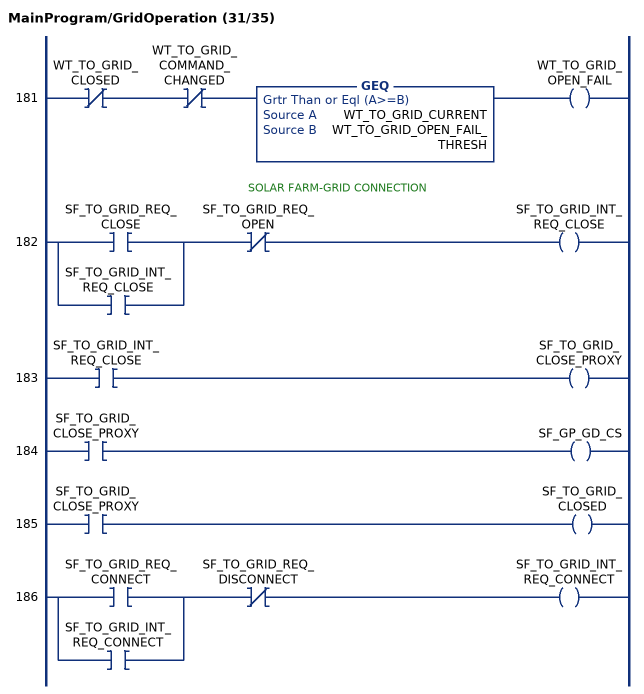
   181: XIO(WT_TO_GRID_CLOSED)XIO(WT_TO_GRID_COMMAND_CHANGED)GEQ(WT_TO_GRID_CURRENT,WT_TO_GRID_OPEN_FAIL_THRESH)OTE(WT_TO_GRID_OPEN_FAIL);
   // SOLAR FARM-GRID CONNECTION
   182: [XIC(SF_TO_GRID_REQ_CLOSE) ,XIC(SF_TO_GRID_INT_REQ_CLOSE) ]XIO(SF_TO_GRID_REQ_OPEN)OTE(SF_TO_GRID_INT_REQ_CLOSE);
   183: XIC(SF_TO_GRID_INT_REQ_CLOSE)OTE(SF_TO_GRID_CLOSE_PROXY);
   184: XIC(SF_TO_GRID_CLOSE_PROXY)OTE(SF_GP_GD_CS);
   185: XIC(SF_TO_GRID_CLOSE_PROXY)OTE(SF_TO_GRID_CLOSED);
   186: [XIC(SF_TO_GRID_REQ_CONNECT) ,XIC(SF_TO_GRID_INT_REQ_CONNECT) ]XIO(SF_TO_GRID_REQ_DISCONNECT)OTE(SF_TO_GRID_INT_REQ_CONNECT);
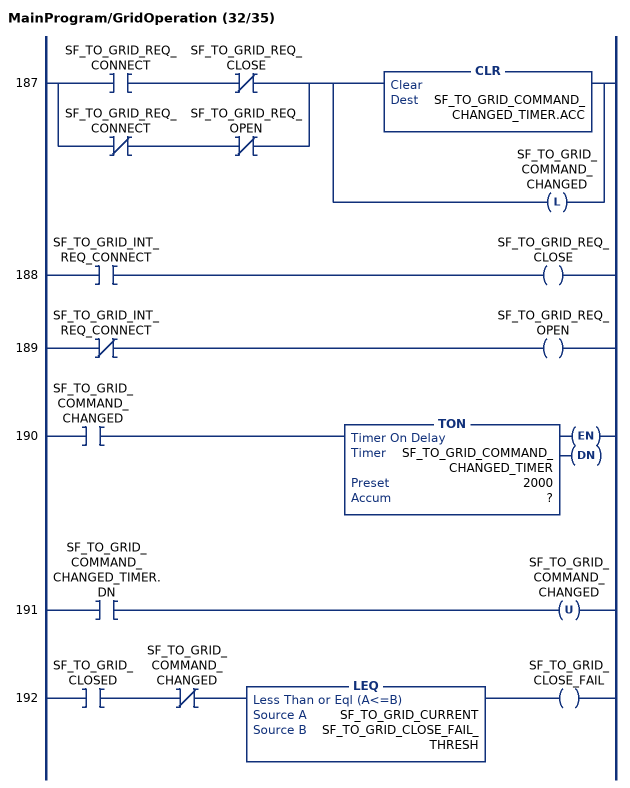
   187: [XIC(SF_TO_GRID_REQ_CONNECT) XIO(SF_TO_GRID_REQ_CLOSE) ,XIO(SF_TO_GRID_REQ_CONNECT) XIO(SF_TO_GRID_REQ_OPEN) ][CLR(SF_TO_GRID_COMMAND_CHANGED_TIMER.ACC) ,OTL(SF_TO_GRID_COMMAND_CHANGED) ];
   188: XIC(SF_TO_GRID_INT_REQ_CONNECT)OTE(SF_TO_GRID_REQ_CLOSE);
   189: XIO(SF_TO_GRID_INT_REQ_CONNECT)OTE(SF_TO_GRID_REQ_OPEN);
   190: XIC(SF_TO_GRID_COMMAND_CHANGED)TON(SF_TO_GRID_COMMAND_CHANGED_TIMER,?,?);
   191: XIC(SF_TO_GRID_COMMAND_CHANGED_TIMER.DN)OTU(SF_TO_GRID_COMMAND_CHANGED);
   192: XIC(SF_TO_GRID_CLOSED)XIO(SF_TO_GRID_COMMAND_CHANGED)LEQ(SF_TO_GRID_CURRENT,SF_TO_GRID_CLOSE_FAIL_THRESH)OTE(SF_TO_GRID_CLOSE_FAIL);
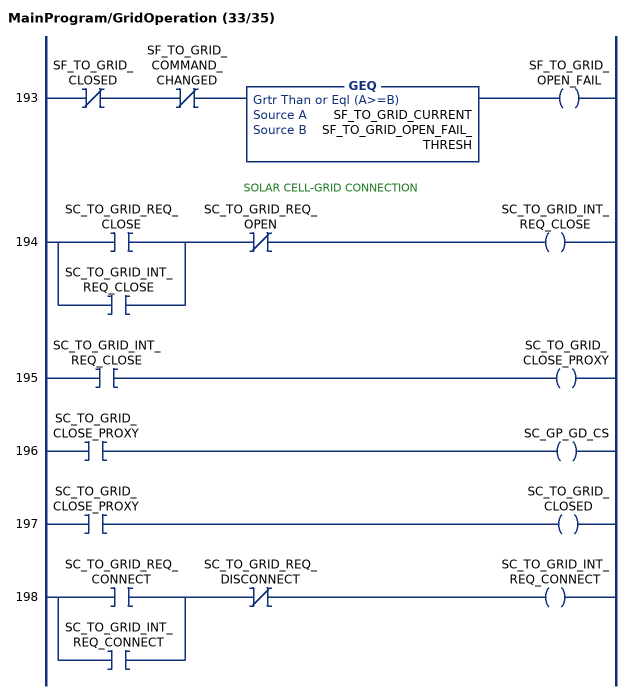
   193: XIO(SF_TO_GRID_CLOSED)XIO(SF_TO_GRID_COMMAND_CHANGED)GEQ(SF_TO_GRID_CURRENT,SF_TO_GRID_OPEN_FAIL_THRESH)OTE(SF_TO_GRID_OPEN_FAIL);
   // SOLAR CELL-GRID CONNECTION
   194: [XIC(SC_TO_GRID_REQ_CLOSE) ,XIC(SC_TO_GRID_INT_REQ_CLOSE) ]XIO(SC_TO_GRID_REQ_OPEN)OTE(SC_TO_GRID_INT_REQ_CLOSE);
   195: XIC(SC_TO_GRID_INT_REQ_CLOSE)OTE(SC_TO_GRID_CLOSE_PROXY);
   196: XIC(SC_TO_GRID_CLOSE_PROXY)OTE(SC_GP_GD_CS);
   197: XIC(SC_TO_GRID_CLOSE_PROXY)OTE(SC_TO_GRID_CLOSED);
   198: [XIC(SC_TO_GRID_REQ_CONNECT) ,XIC(SC_TO_GRID_INT_REQ_CONNECT) ]XIO(SC_TO_GRID_REQ_DISCONNECT)OTE(SC_TO_GRID_INT_REQ_CONNECT);
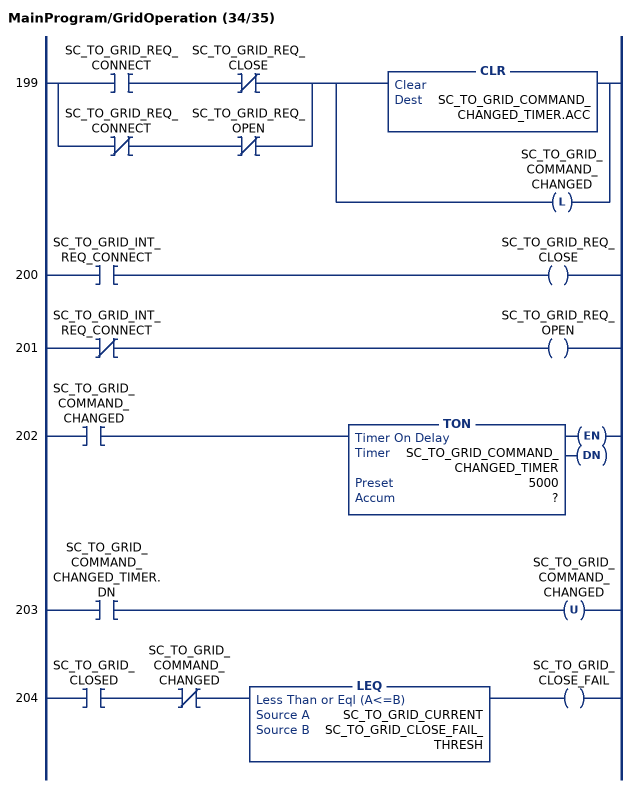
   199: [XIC(SC_TO_GRID_REQ_CONNECT) XIO(SC_TO_GRID_REQ_CLOSE) ,XIO(SC_TO_GRID_REQ_CONNECT) XIO(SC_TO_GRID_REQ_OPEN) ][CLR(SC_TO_GRID_COMMAND_CHANGED_TIMER.ACC) ,OTL(SC_TO_GRID_COMMAND_CHANGED) ];
   200: XIC(SC_TO_GRID_INT_REQ_CONNECT)OTE(SC_TO_GRID_REQ_CLOSE);
   201: XIO(SC_TO_GRID_INT_REQ_CONNECT)OTE(SC_TO_GRID_REQ_OPEN);
   202: XIC(SC_TO_GRID_COMMAND_CHANGED)TON(SC_TO_GRID_COMMAND_CHANGED_TIMER,?,?);
   203: XIC(SC_TO_GRID_COMMAND_CHANGED_TIMER.DN)OTU(SC_TO_GRID_COMMAND_CHANGED);
   204: XIC(SC_TO_GRID_CLOSED)XIO(SC_TO_GRID_COMMAND_CHANGED)LEQ(SC_TO_GRID_CURRENT,SC_TO_GRID_CLOSE_FAIL_THRESH)OTE(SC_TO_GRID_CLOSE_FAIL);
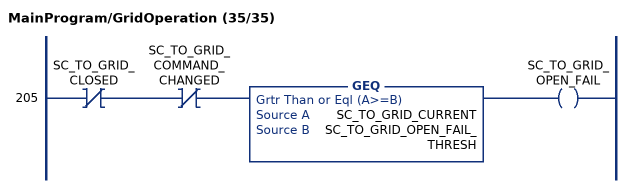
   205: XIO(SC_TO_GRID_CLOSED)XIO(SC_TO_GRID_COMMAND_CHANGED)GEQ(SC_TO_GRID_CURRENT,SC_TO_GRID_OPEN_FAIL_THRESH)OTE(SC_TO_GRID_OPEN_FAIL);
END_ROUTINE
